// States for state machine used in `DynamicStringBuffer.PersistToFile`
{attribute 'qualified_only'}
{attribute 'strict'}
TYPE INTERNAL PersistToFileState :
(
	Idle := 0,
	OpenFile,
	GetStringFromFifo,
	AppendDataToFile,
	CloseFile
);
END_TYPE

(* stored: Version 1.1.0.1
   DUT PersistToFileState: Id {f165e319-464b-4a7b-a486-84fad9259575} *)
